(* IEC 61131-3 sources: volt/packages/volt-lsp-iec/test-corpus/bakon-nano/Device/Plc Logic/Application/Library Manager/CAA Async Manager, 37 files *)

(* ---- ASM_CURRENT_MAX.dut ---- *)
TYPE ASM_CURRENT_MAX :
STRUCT
	CURRENT : CAA.COUNT;
	MAXIMUM : CAA.COUNT;
END_STRUCT
END_TYPE

(* ---- ASM_IWORKER.dut ---- *)
TYPE ASM_IWORKER :
STRUCT
	PFEXEC : CAA.PVOID;
	PFABORT : CAA.PVOID;
	PFGETSTATE : CAA.PVOID;
	PFDISPOSE : CAA.PVOID;
	PFGETPARAMSIZE : CAA.PVOID;
END_STRUCT
END_TYPE

(* ---- ASM_STATE.dut ---- *)
TYPE ASM_STATE :
STRUCT
	EERROR : INT;
	ESTATE : JOB_STATE;
	USIPROGRESS : USINT;
END_STRUCT
END_TYPE

(* ---- ERROR.dut ---- *)
TYPE ERROR :
(
	NO_ERROR := 0,
	FIRST_ERROR := 5800,
	HANDLE_INVALID := 5802,
	WRONG_ARGUMENT := 5803,
	NO_WORKER := 5804,
	WORKER_REGISTERED := 5805,
	ID_INVALID := 5806,
	WRONG_STATE := 5807,
	STATE_INVALID := 5808,
	NO_MEMORY := 5809,
	FIRST_MF := 5820,
	LAST_ERROR := 5850
);
END_TYPE

(* ---- IWORKER.dut ---- *)
TYPE IWORKER : ASM_IWORKER;
END_TYPE

(* ---- JOB_STATE.dut ---- *)
TYPE JOB_STATE :
(
	DORMANT := 0,
	BUSY := 1,
	DONE := 2,
	ABORTED := 3,
	STATE_ERROR
);
END_TYPE

(* ---- STATE.dut ---- *)
TYPE STATE : ASM_STATE;
END_TYPE

(* ---- RSHANDLING.gvl ---- *)
VAR_GLOBAL
	G_JOBCLASS : JobClass;
END_VAR

(* ---- VERSIONCONSTANTS.gvl ---- *)
VAR_GLOBAL
	GC_BYVERSION : BYTE := 1;
	GC_BYVERSION_1 : BYTE := 0;
END_VAR

(* ---- _JOBABORT.pou ---- *)
FUNCTION _JOBABORT : ERROR
VAR_INPUT
	HJOB : CAA.HANDLE;
END_VAR
END_FUNCTION

(* ---- _JOBCLOSE.pou ---- *)
FUNCTION _JOBCLOSE : ERROR
VAR_INPUT
	HJOB : CAA.HANDLE;
END_VAR
END_FUNCTION

(* ---- _JOBEXECUTE.pou ---- *)
FUNCTION _JOBEXECUTE : ERROR
VAR_INPUT
	HJOB : CAA.HANDLE;
END_VAR
END_FUNCTION

(* ---- _JOBGETID.pou ---- *)
FUNCTION _JOBGETID : UDINT
VAR_INPUT
	HJOB : CAA.HANDLE;
	PEERROR : POINTER TO ERROR;
END_VAR
END_FUNCTION

(* ---- _JOBGETNUMOFJOBS.pou ---- *)
FUNCTION _JOBGETNUMOFJOBS : ERROR
VAR_IN_OUT
	NUMOFJOBS : ASM_CURRENT_MAX;
	NUMOFWORKERS : ASM_CURRENT_MAX;
END_VAR
END_FUNCTION

(* ---- _JOBGETPARAMS.pou ---- *)
FUNCTION _JOBGETPARAMS : CAA.PVOID
VAR_INPUT
	HJOB : CAA.HANDLE;
	PEERROR : POINTER TO ERROR;
END_VAR
END_FUNCTION

(* ---- _JOBGETSTATE.pou ---- *)
FUNCTION _JOBGETSTATE : ERROR
VAR_INPUT
	HJOB : CAA.HANDLE;
	PSTATEJOB : POINTER TO ASM_STATE;
END_VAR
END_FUNCTION

(* ---- _JOBOPEN.pou ---- *)
FUNCTION _JOBOPEN : CAA.HANDLE
VAR_INPUT
	UDIID : UDINT;
	PEERROR : POINTER TO ERROR;
END_VAR
END_FUNCTION

(* ---- _JOBOPENEX.pou ---- *)
FUNCTION _JOBOPENEX : CAA.HANDLE
VAR_INPUT
	UDIID : UDINT;
	PPARAMS : CAA.PVOID;
	PEERROR : POINTER TO ERROR;
END_VAR
END_FUNCTION

(* ---- _JOBRESET.pou ---- *)
FUNCTION _JOBRESET : ERROR
VAR_INPUT
	HJOB : CAA.HANDLE;
END_VAR
END_FUNCTION

(* ---- _JOBSETSTATE.pou ---- *)
FUNCTION _JOBSETSTATE : ERROR
VAR_INPUT
	HJOB : CAA.HANDLE;
	STATEJOB : ASM_STATE;
END_VAR
END_FUNCTION

(* ---- _WORKERREGISTER.pou ---- *)
FUNCTION _WORKERREGISTER : ERROR
VAR_INPUT
	UDIID : UDINT;
	PWITF : POINTER TO ASM_IWORKER;
END_VAR
END_FUNCTION

(* ---- _WORKERUNREGISTER.pou ---- *)
FUNCTION _WORKERUNREGISTER : ERROR
VAR_INPUT
	UDIID : UDINT;
END_VAR
END_FUNCTION

(* ---- GETSUPPLIERVERSION.pou ---- *)
FUNCTION GETSUPPLIERVERSION : WORD
END_FUNCTION

(* ---- JOBABORT.pou ---- *)
FUNCTION JOBABORT : ERROR
VAR_INPUT
	HJOB : CAA.HANDLE;
END_VAR
END_FUNCTION

(* ---- JOBCLOSE.pou ---- *)
FUNCTION JOBCLOSE : ERROR
VAR_INPUT
	HJOB : CAA.HANDLE;
END_VAR
END_FUNCTION

(* ---- JOBEXECUTE.pou ---- *)
FUNCTION JOBEXECUTE : ERROR
VAR_INPUT
	HJOB : CAA.HANDLE;
END_VAR
END_FUNCTION

(* ---- JOBGETID.pou ---- *)
FUNCTION JOBGETID : UDINT
VAR_INPUT
	HJOB : CAA.HANDLE;
	PEERROR : POINTER TO ERROR;
END_VAR
END_FUNCTION

(* ---- JOBGETNUMOFJOBS.pou ---- *)
FUNCTION JOBGETNUMOFJOBS : ERROR
VAR_INPUT
	NUMOFJOBS : POINTER TO ASM_CURRENT_MAX;
	NUMOFWORKERS : POINTER TO ASM_CURRENT_MAX;
END_VAR
END_FUNCTION

(* ---- JOBGETPARAMS.pou ---- *)
FUNCTION JOBGETPARAMS : CAA.PVOID
VAR_INPUT
	HJOB : CAA.HANDLE;
	PEERROR : POINTER TO ERROR;
END_VAR
END_FUNCTION

(* ---- JOBGETSTATE.pou ---- *)
FUNCTION JOBGETSTATE : ERROR
VAR_INPUT
	HJOB : CAA.HANDLE;
	PSTATEJOB : POINTER TO STATE;
END_VAR
END_FUNCTION

(* ---- JOBOPEN.pou ---- *)
FUNCTION JOBOPEN : CAA.HANDLE
VAR_INPUT
	UDIID : UDINT;
	PEERROR : POINTER TO ERROR;
END_VAR
END_FUNCTION

(* ---- JOBOPENEX.pou ---- *)
FUNCTION JOBOPENEX : CAA.HANDLE
VAR_INPUT
	UDIID : UDINT;
	PPARAMS : CAA.PVOID;
	PEERROR : POINTER TO ERROR;
END_VAR
END_FUNCTION

(* ---- JOBRESET.pou ---- *)
FUNCTION JOBRESET : ERROR
VAR_INPUT
	HJOB : CAA.HANDLE;
END_VAR
END_FUNCTION

(* ---- JOBSETSTATE.pou ---- *)
FUNCTION JOBSETSTATE : ERROR
VAR_INPUT
	HJOB : CAA.HANDLE;
	STATEJOB : ASM_STATE;
END_VAR
END_FUNCTION

(* ---- WORKERREGISTER.pou ---- *)
FUNCTION WORKERREGISTER : ERROR
VAR_INPUT
	UDIID : UDINT;
	PWITF : POINTER TO ASM_IWORKER;
END_VAR
END_FUNCTION

(* ---- WORKERUNREGISTER.pou ---- *)
FUNCTION WORKERUNREGISTER : ERROR
VAR_INPUT
	UDIID : UDINT;
END_VAR
END_FUNCTION

(* ---- JOBCLASS.pou ---- *)
FUNCTION_BLOCK JOBCLASS EXTENDS RSMClass
END_FUNCTION_BLOCK

METHOD CLOSE : RSM.ERROR
VAR_INPUT
	HHANDLE : CAA.HANDLE;
END_VAR
END_METHOD
